PROGRAM OOP_MAIN
VAR
	FuzzyLogicController:FB_FIS_oop;
	
END_VAR

END_PROGRAM

(* stored: Version 1.1.0.1, ProductVersion 3.1.4024.6
   POU OOP_MAIN: Id {290bccff-ad29-4b05-ad7e-0058b322cbac}, SpecialFunc None *)
